SUBAPPLICATION Softkey_Aux_IE (* SoftKey ODER AUX-Zuweisung (Joystick) aktiviert -> 1 gemeinsames IND-Event (SK_PRESSED bzw. AuxEnabled fest verdrahtet - die einzig sinnvolle 'aktiviert'-Bedeutung fuer eine Merge-Anwendung). Analog zu Softkey_Aux_IXA_TO_Remote_WRITE (Dauerzustand-ODER), aber fuer den diskreten Event-Kanal - kollidiert daher nicht mit einer bereits bestehenden Softkey_IXA/Aux_IXA-Dauerzustand-Abonnierung auf demselben Objekt (2 verschiedene Subscription-Typen). *)
  (* Standard: 61499-2 *)
  (* Version 1.0, 2026-09-11, Franz Höpfinger, initial implementation *)
  PACKAGE MyLib::sys;
  IMPORT isobus::UT::io::Softkey::SoftKeyActivationCode::SK_PRESSED;
  IMPORT isobus::UT::io::Auxiliary::IN::AuxiliaryState::AuxEnabled;
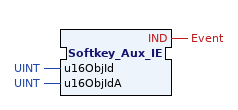
  EVENT_OUTPUT
    IND; (* Feuert wenn SoftKey (SK_PRESSED) ODER Aux (AuxEnabled) aktiviert wird *)
  END_EVENT
  VAR_INPUT
    u16ObjId : UINT; (* Object ID SoftKey *)
    u16ObjIdA : UINT; (* Object ID AuxFunction2 *)
  END_VAR
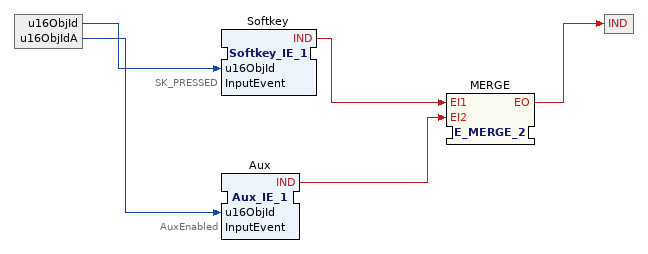
  FBS
    MERGE : iec61499::events::E_MERGE_2;
  END_FBS
  SUBAPPS
    Softkey : MyLib::sys::Softkey_IE_1(InputEvent := SK_PRESSED);
    Aux : MyLib::sys::Aux_IE_1(InputEvent := AuxEnabled);
  END_SUBAPPS
  EVENT_CONNECTIONS
    Softkey.IND TO MERGE.EI1;
    Aux.IND TO MERGE.EI2;
    MERGE.EO TO IND;
  END_CONNECTIONS
  DATA_CONNECTIONS
    u16ObjId TO Softkey.u16ObjId;
    u16ObjIdA TO Aux.u16ObjId;
  END_CONNECTIONS
END_SUBAPPLICATION
